FUNCTION_BLOCK AlarmServer
VAR CONSTANT
	nrAlarms 			: UINT := 2000;
	sTable 				: STRING:= '"public"."datatypes"'; // Important to have extra " " around both DBname and table name.
	DBID				: UINT	:=1;
	
	//For read Method
	OrderByColumn		: UINT	:=1; 
	StartIndex			: UINT	:=0;
END_VAR
VAR
	init 				: BOOL:= TRUE;
	ColumnNames     	: ARRAY[0..4] OF STRING(50); // Must be set to 50 char!
	dataReturned 		: ARRAY[0..9] OF Alarms; // Array of the numbers of rows you want to store. 
END_VAR
VAR PERSISTENT
	AlarmData			: ARRAY [0..nrAlarms] OF Alarms;
	iValueChanged 		: INT;
	irowSelected		: INT;
	bAckAlarm 			: BOOL;
	bAckAllAlarms 		: BOOL;
	bClearAllAlarms 	: BOOL;
END_VAR

// First run, init stuff needed to work
IF init THEN
	// Set columnnames -- Must be the same as in DB
	ColumnNames[0] := '_name';
	ColumnNames[1] := '_dint';
	ColumnNames[2] := '_real';
	ColumnNames[3] := '_lreal';
	ColumnNames[4] := '_date';
	
	init:= FALSE;
END_IF



IF(bAckAlarm) THEN
	bAckAlarm:= FALSE;
	AckAlarm(iRow:= irowSelected);
END_IF

IF(bAckAllAlarms) THEN
	bAckAllAlarms:= FALSE;
	AckAllAlarms();
END_IF

IF(bClearAllAlarms) THEN
	bClearAllAlarms:= FALSE;
	ClearAllAlarms();
END_IF

METHOD PUBLIC AckAlarm : BOOL
VAR_INPUT
	iRow: INT;
END_VAR

VAR
	i: UINT;
	actDC : T_DCTIME64;
    sAct  : STRING;
END_VAR
actDC := F_GetActualDcTime64();
sAct  := DCTIME64_TO_STRING( actDC );

AlarmData[iRow].bIsAcknowledged:=  TRUE;
AlarmData[iRow].tAcknowlegedTime :=  sAct;


// Update variable for valuechange event
iValueChanged:= iValueChanged +1;
// Always add to DB
//AddToDb(AlarmData[i]);
END_METHOD

METHOD PUBLIC AckAllAlarms : BOOL
VAR
	i: UINT;
	actDC : T_DCTIME64;
    sAct  : STRING;
	Alarm: Alarms;
END_VAR
actDC := F_GetActualDcTime64();
sAct  := DCTIME64_TO_STRING( actDC );

FOR i:=0 TO nrAlarms BY 1 DO
	
	IF AlarmData[i].bIsUsed THEN
		
		AlarmData[i].bIsAcknowledged:=  TRUE;
		AlarmData[i].tAcknowlegedTime :=  sAct;
		// Always add to DB before removing alarm in server
		AddToDb(Alarm);
	END_IF
	
END_FOR

// Update variable for valuechange event
iValueChanged:= iValueChanged +1;
END_METHOD

METHOD PUBLIC AddToDb : BOOL
VAR_INPUT
	Alarm: Alarms;
END_VAR
VAR
	fbPLCDBWrite    	: FB_PLCDBWriteEvt(sNetID := '', tTimeout := T#5S);
	tcMessage       	: I_TcMessage;	
END_VAR
// Write one record to Database 
// Call Functionblock
IF fbPLCDBWrite.WriteStruct(
	hDBID:= DBID, 
	sTableName:= sTable, 
	pRecord:= ADR(Alarm), 
	cbRecord:= SIZEOF(Alarm), 
	pColumnNames:= ADR(ColumnNames) , 
	cbColumnNames:= SIZEOF(ColumnNames))
THEN
	IF fbPLCDBWrite.bError THEN
		tcMessage := fbPLCDBWrite.ipTcResult;
	END_IF
END_IF
END_METHOD

METHOD PUBLIC ClearAllAlarms : BOOL
VAR
	Alarm: Alarms;
	i: UINT;
	actDC : T_DCTIME64;
    sAct  : STRING;
	
END_VAR
actDC := F_GetActualDcTime64();
sAct  := DCTIME64_TO_STRING( actDC );

FOR i:=0 TO nrAlarms BY 1 DO
	
	IF AlarmData[i].bIsAcknowledged = TRUE THEN
		AlarmData[i].tClearedTime :=  sAct;
		// Always add to DB before removing alarm in server
		AddToDb(AlarmData[i]);
		AlarmData[i]:= Alarm;
	END_IF
	
END_FOR
// Update variable for valuechange event
iValueChanged:= iValueChanged +1;
END_METHOD

METHOD PUBLIC NewAlarm : BOOL
VAR_INPUT
	sName: STRING;
	sAlarmText: STRING;	
END_VAR
VAR
	Alarm: Alarms;
	i: UINT;
	bAlarmExists : BOOL;

	actDC : T_DCTIME64;
    sAct  : STRING;
END_VAR
Alarm.sName := sName;
Alarm.sAlarmText := sAlarmText; 
Alarm.bIsActive := TRUE;
Alarm.bIsUsed := TRUE;

actDC := F_GetActualDcTime64();
sAct  := DCTIME64_TO_STRING( actDC );

Alarm.tActiveStartTime :=  sAct;

FOR i:=0 TO nrAlarms BY 1 DO
	
	IF (AlarmData[i].bIsUsed = TRUE AND AlarmData[i].sName = sName) THEN
		AlarmData[i].uiRepeatCount := AlarmData[i].uiRepeatCount + 1;
		AlarmData[i].tActiveStartTime := Alarm.tActiveStartTime;
		AlarmData[i].tAcknowlegedTime := '';
		AlarmData[i].bIsAcknowledged := FALSE;
		bAlarmExists:= TRUE;
		EXIT;
	END_IF
	
END_FOR
 
IF bAlarmExists = FALSE THEN
	
	FOR i:=0 TO SIZEOF(AlarmData) - 1 BY 1 DO
		
		IF (AlarmData[i].bIsUsed = FALSE) THEN
			AlarmData[i] := Alarm;
			EXIT;	
		END_IF
		
	END_FOR
END_IF

// Update variable for valuechange event
iValueChanged:= iValueChanged +1;
// Always add to DB
//AddToDb(Alarm);
END_METHOD

METHOD PUBLIC ReadFromDB : BOOL
VAR_INPUT
	NrOfRows 			: UINT:=10;
END_VAR
VAR
	fbPLCDBRead    		: FB_PLCDBReadEvt (sNetID := '', tTimeout := T#5S);
    tcMessage	     	: I_TcMessage;
	
END_VAR
//	Read rows from the db.  	 
IF fbPLCDBRead.ReadStruct(
	hDBID:= DBID, 
	sTableName:= sTable, 
	pColumnNames:= ADR(ColumnNames), 
	cbColumnNames:= SIZEOF(ColumnNames), 
	sOrderByColumn:= ColumnNames[OrderByColumn], 
	eOrderType:= E_OrderType.ASC, 
	nStartIndex:= StartIndex, 
	nRecordCount:= NrOfRows, 
	pData:= ADR(dataReturned), 
	cbData:= SIZEOF(dataReturned))
THEN

	IF fbPLCDBRead.bError THEN
		tcMessage:= fbPLCDBRead.ipTcResult;
	END_IF
END_IF
//
END_METHOD

END_FUNCTION_BLOCK

(* stored: Version 1.1.0.1, ProductVersion 3.1.4024.9
   POU AlarmServer: Id {3d2cc0da-a4c3-43eb-906a-300187b5ba2d}, SpecialFunc None
   Method AckAlarm: Id {3998354c-f7a9-4477-9dd1-1e1dd91ff7c6}
   Method AckAllAlarms: Id {d37e7b81-01f0-40d0-83bf-50bc651716c7}
   Method AddToDb: Id {bacaf7d5-fbb6-464d-b066-8afef850f3b6}
   Method ClearAllAlarms: Id {1ecd57a5-9500-4f9c-86c4-237a9ec07bd0}
   Method NewAlarm: Id {ff3e33e4-bc96-4829-912e-fd21b8af1018}
   Method ReadFromDB: Id {7e1f915b-3b34-44c6-a7c3-63f4fb4fd38f} *)
